// TIA Portal V17 export
// export: Created 2022-07-28T18:02:47.0789834Z, ExportSetting None, DisplayName Totally Integrated Automation Portal, DisplayVersion V17, DisplayName TIA Portal Openness, DisplayVersion V17, DisplayName TIA Portal Teamcenter Gateway, DisplayVersion V17, DisplayName TIA Portal Version Control Interface, DisplayVersion V17, DisplayName TIA Portal Test Suite Advanced, DisplayVersion V17, DisplayName SINAMICS Startdrive Advanced, DisplayVersion V17, DisplayName SINAMICS DCC, DisplayVersion V17, DisplayName SINAMICS Startdrive G130, G150, S120, S150, SINAMICS MV, S210, DisplayVersion V17, DisplayName SINAMICS Startdrive G110M, G120, G120C, G120D, G120P, G115D, DisplayVersion V17, DisplayName STEP 7 Professional, DisplayVersion V17, DisplayName SIMATIC Energy Suite, DisplayVersion V17, DisplayName STEP 7 CFC, DisplayVersion V17, DisplayName STEP 7 Safety, DisplayVersion V17, DisplayName WinCC Advanced / Unified PC, DisplayVersion V17, DisplayName SIMATIC Visualization Architect, DisplayVersion V17
FUNCTION "Outputs_FC" : Void   // FC14, SCL
{ S7_Optimized_Access := 'TRUE' }
// stored: SetENOAutomatically false
BEGIN
   REGION (ID = 1) Витратомір пари на нову рафінацію Steam Flowmeter New
       //Тип елемента: Аналоговий витратомір
       //Параметри давача: Scale=; 4-20mA; Analog = 0 - 27648;
       //Одиниці вимірювання: m3/h
       //Додаткова інформація: SITRANS FX330 / 7ME2610-3LD00-0AA0-Z

   END_REGION

   REGION (ID = 2) Витратомір пари на стару рафінацію Steam Flowmeter Old
       //Тип елемента: Аналоговий витратомір
       //Параметри давача: Scale=; 4-20mA; Analog = 0 - 27648;
       //Одиниці вимірювання: m3/h
       //Додаткова інформація: SITRANS FX330 / 7ME2610-3LD00-0AA0-Z

   END_REGION

   REGION (ID = 3) Перетворювач тиску обор.води PTНГр
       //Тип елемента: Аналоговий сигнал
       //Параметри давача: Scale=0-10bar; 4-20mA; Analog = 0 - 27648;
       //Одиниці вимірювання: bar
       //Додаткова інформація: 

   END_REGION

   REGION (ID = 4) Перетворювач температури вих.води ХМ1 ТТW1011
       //Тип елемента: Аналоговий сигнал
       //Параметри давача: Scale=0-150C; 4-20mA; Analog = 0 - 27648;
       //Одиниці вимірювання: C
       //Додаткова інформація: 

   END_REGION

   REGION (ID = 5) Перетворювач температури вих.води ХМ2 TT811
       //Тип елемента: Аналоговий сигнал
       //Параметри давача: Scale=0-150C; 4-20mA; Analog = 0 - 27648;
       //Одиниці вимірювання: C
       //Додаткова інформація: 

   END_REGION

   REGION (ID = 6) Перетворювач тиску (рівень басейну градирні 1) LTБ1Гр
       //Тип елемента: Аналоговий сигнал
       //Параметри давача: Scale=0-0.25bar; 4-20mA; Analog = 0 - 27648;
       //Одиниці вимірювання: м
       //Додаткова інформація: 

   END_REGION

   REGION (ID = 7) Перетворювач тиску (рівень басейну градирні 2) LTБ2Гр
       //Тип елемента: Аналоговий сигнал
       //Параметри давача: Scale=0-0.25bar; 4-20mA; Analog = 0 - 27648;
       //Одиниці вимірювання: м
       //Додаткова інформація: 

   END_REGION

   REGION (ID = 8) Аналоговий сигнал від AirForce 1 G1
       //Тип елемента: Аналоговий сигнал
       //Параметри давача: Scale= ; 4-20mA; Analog = 0 - 27648;
       //Одиниці вимірювання: 
       //Додаткова інформація: 

   END_REGION

   REGION (ID = 9) Аналоговий сигнал від AirForce 2 G1
       //Тип елемента: Аналоговий сигнал
       //Параметри давача: Scale= ; 4-20mA; Analog = 0 - 27648;
       //Одиниці вимірювання: 
       //Додаткова інформація: 

   END_REGION

   REGION (ID = 10) Аналоговий сигнал від AirForce 3 G1
       //Тип елемента: Аналоговий сигнал
       //Параметри давача: Scale= ; 4-20mA; Analog = 0 - 27648;
       //Одиниці вимірювання: 
       //Додаткова інформація: 

   END_REGION

   REGION (ID = 11) Аналоговий сигнал від AirForce 4 G1
       //Тип елемента: Аналоговий сигнал
       //Параметри давача: Scale= ; 4-20mA; Analog = 0 - 27648;
       //Одиниці вимірювання: 
       //Додаткова інформація: 

   END_REGION

   REGION (ID = 12) Аналоговий сигнал від AirForce 5 G1
       //Тип елемента: Аналоговий сигнал
       //Параметри давача: Scale= ; 4-20mA; Analog = 0 - 27648;
       //Одиниці вимірювання: 
       //Додаткова інформація: 

   END_REGION

   REGION (ID = 13) Аналоговий сигнал від AirForce 6 G1
       //Тип елемента: Аналоговий сигнал
       //Параметри давача: Scale= ; 4-20mA; Analog = 0 - 27648;
       //Одиниці вимірювання: 
       //Додаткова інформація: 

   END_REGION

   REGION (ID = 14) Перетворювач тиску (рівень ємності конденсату) LT R46
       //Тип елемента: Аналоговий сигнал
       //Параметри давача: Scale=0-0.4bar; 4-20mA; Analog = 0 - 27648;
       //Одиниці вимірювання: м
       //Додаткова інформація: 

   END_REGION

   REGION (ID = 15) Температура конденсату TT R46
       //Тип елемента: Аналоговий сигнал
       //Параметри давача: Scale=0-150C; 4-20mA; Analog = 0 - 27648;
       //Одиниці вимірювання: C
       //Додаткова інформація: 

   END_REGION

   REGION (ID = 16) Тиск повітря 1 PT AirLow
       //Тип елемента: Аналоговий сигнал
       //Параметри давача: Scale=0-10bar; 4-20mA; Analog = 0 - 27648;
       //Одиниці вимірювання: bar
       //Додаткова інформація: 

   END_REGION

   REGION (ID = 17) Тиск повітря 2 PT AirHigh
       //Тип елемента: Аналоговий сигнал
       //Параметри давача: Scale=0-10bar; 4-20mA; Analog = 0 - 27648;
       //Одиниці вимірювання: bar
       //Додаткова інформація: 

   END_REGION

   REGION (ID = 18) Тиск газу PT Gas
       //Тип елемента: Аналоговий сигнал
       //Параметри давача: Scale= ;4-20ma; Analog = 0 - 27648;
       //Одиниці вимірювання: 
       //Додаткова інформація: 

   END_REGION

   REGION (ID = 19) Тиск азоту PT Nitrogen
       //Тип елемента: Аналоговий сигнал
       //Параметри давача: Scale= ;4-20ma; Analog = 0 - 27648;
       //Одиниці вимірювання: 
       //Додаткова інформація: 

   END_REGION

   REGION (ID = 20) Тиск води осмотичної PT W10_1
       //Тип елемента: Аналоговий сигнал
       //Параметри давача: Scale=0-6bar; 4-20mA; Analog = 0 - 27648;
       //Одиниці вимірювання: bar
       //Додаткова інформація: 

   END_REGION

   REGION (ID = 21) Тиск води технічної PT water
       //Тип елемента: Аналоговий сигнал
       //Параметри давача: Scale=0-6bar; 4-20mA; Analog = 0 - 27648;
       //Одиниці вимірювання: bar
       //Додаткова інформація: 

   END_REGION

   REGION (ID = 22) Тиск пари 1 PT steam 1
       //Тип елемента: Аналоговий сигнал
       //Параметри давача: Scale= ;4-20ma; Analog = 0 - 27648;
       //Одиниці вимірювання: 
       //Додаткова інформація: 

   END_REGION

   REGION (ID = 23) Тиск пари 2 PT steam 2
       //Тип елемента: Аналоговий сигнал
       //Параметри давача: Scale= ;4-20ma; Analog = 0 - 27648;
       //Одиниці вимірювання: 
       //Додаткова інформація: 

   END_REGION

   REGION (ID = 24) Тиск пари 3 PT steam 3
       //Тип елемента: Аналоговий сигнал
       //Параметри давача: Scale= ;4-20ma; Analog = 0 - 27648;
       //Одиниці вимірювання: 
       //Додаткова інформація: 

   END_REGION

   REGION (ID = 25) Тиск теплоносія 1 PT coolant 1
       //Тип елемента: Аналоговий сигнал
       //Параметри давача: Scale= ;4-20ma; Analog = 0 - 27648;
       //Одиниці вимірювання: 
       //Додаткова інформація: 

   END_REGION

   REGION (ID = 26) Тиск теплоносія 2 PT coolant 2
       //Тип елемента: Аналоговий сигнал
       //Параметри давача: Scale= ;4-20ma; Analog = 0 - 27648;
       //Одиниці вимірювання: 
       //Додаткова інформація: 

   END_REGION

   REGION (ID = 27) Температура теплоносія 1 TT coolant 1
       //Тип елемента: Аналоговий сигнал
       //Параметри давача: Scale=0-150C; 4-20mA; Analog = 0 - 27648;
       //Одиниці вимірювання: C
       //Додаткова інформація: 

   END_REGION

   REGION (ID = 28) Температура теплоносія 2 TT coolant 2
       //Тип елемента: Аналоговий сигнал
       //Параметри давача: Scale=0-150C; 4-20mA; Analog = 0 - 27648;
       //Одиниці вимірювання: C
       //Додаткова інформація: 

   END_REGION

   REGION (ID = 29) Перетворювач тиску подачі  кислоти PT PW579CA
       //Тип елемента: Аналоговий сигнал
       //Параметри давача: Scale=0-6bar; 4-20mA; Analog = 0 - 27648;
       //Одиниці вимірювання: bar
       //Додаткова інформація: 

   END_REGION

   REGION (ID = 30) Рівень в ємності лимонної кислоти LT PW579CA
       //Тип елемента: Аналоговий сигнал
       //Параметри давача: Scale=0-0.1bar; 4-20mA; Analog = 0 - 27648;
       //Одиниці вимірювання: м
       //Додаткова інформація: 

   END_REGION

   REGION (ID = 31) Перетворювач тиску подачі  лугу PT PW579NA
       //Тип елемента: Аналоговий сигнал
       //Параметри давача: Scale=0-6bar; 4-20mA; Analog = 0 - 27648;
       //Одиниці вимірювання: bar
       //Додаткова інформація: 

   END_REGION

   REGION (ID = 32) Перетворювач тиску (рівень води в ємності) LT W10 OW
       //Тип елемента: Аналоговий сигнал
       //Параметри давача: Scale=0-0.25bar; 4-20mA; Analog = 0 - 27648;
       //Одиниці вимірювання: м
       //Додаткова інформація: 

   END_REGION

   REGION (ID = 33) Температура води охолодження дублюючого насоса TT P822 2
       //Тип елемента: Аналоговий сигнал
       //Параметри давача: Scale= ; 4-20mA; Analog = 0 - 27648;
       //Одиниці вимірювання: C
       //Додаткова інформація: 

   END_REGION

   REGION (ID = 34) Рівень води в ємності LT W0 W
       //Тип елемента: Аналоговий сигнал
       //Параметри давача: Scale=0-0.25bar; 4-20mA; Analog = 0 - 27648;
       //Одиниці вимірювання: м
       //Додаткова інформація: 

   END_REGION

   REGION (ID = 35) Перетворювач тиску технологічної води PT PW0 W
       //Тип елемента: Аналоговий сигнал
       //Параметри давача: Scale=0-10bar; 4-20mA; Analog = 0 - 27648;
       //Одиниці вимірювання: bar
       //Додаткова інформація: 

   END_REGION

   REGION (ID = 36) Дискретний сигнал від AirForce 1 G1
       //Тип елемента: Дискретний сигнал
       //Параметри давача: Info;NO;
       //Додаткова інформація: 

   END_REGION

   REGION (ID = 37) Дискретний сигнал від AirForce 2 G1
       //Тип елемента: Дискретний сигнал
       //Параметри давача: Info;NO;
       //Додаткова інформація: 

   END_REGION

   REGION (ID = 38) Дискретний сигнал від AirForce 3 G1
       //Тип елемента: Дискретний сигнал
       //Параметри давача: Info;NO;
       //Додаткова інформація: 

   END_REGION

   REGION (ID = 39) Дискретний сигнал від AirForce 4 G1
       //Тип елемента: Дискретний сигнал
       //Параметри давача: Info;NO;
       //Додаткова інформація: 

   END_REGION

   REGION (ID = 40) Дискретний сигнал від AirForce 5 G1
       //Тип елемента: Дискретний сигнал
       //Параметри давача: Info;NO;
       //Додаткова інформація: 

   END_REGION

   REGION (ID = 41) Контроль роботи холодильної машини 1 - робота W1011
       //Тип елемента: Дискретний сигнал
       //Параметри давача: Info;NO;
       //Додаткова інформація: 

   END_REGION

   REGION (ID = 42) Контроль роботи холодильної машини 1 - аварія W1011
       //Тип елемента: Дискретний сигнал
       //Параметри давача: Err;NO;
       //Додаткова інформація: 

   END_REGION

   REGION (ID = 43) Контроль роботи холодильної машини 2 - робота 811
       //Тип елемента: Дискретний сигнал
       //Параметри давача: Info;NO;
       //Додаткова інформація: 

   END_REGION

   REGION (ID = 44) Контроль роботи холодильної машини 2 - аварія 811
       //Тип елемента: Дискретний сигнал
       //Параметри давача: Err;NO;
       //Додаткова інформація: 

   END_REGION

   REGION (ID = 45) Парогенератор і бойлерна - робота DI7
       //Тип елемента: Дискретний сигнал
       //Параметри давача: Info;NO;
       //Додаткова інформація: 

   END_REGION

   REGION (ID = 46) Парогенератор і бойлерна - аварія DI7
       //Тип елемента: Дискретний сигнал
       //Параметри давача: Err;NC;
       //Додаткова інформація: 

   END_REGION

   REGION (ID = 47) Парогенератор і бойлерна - загазованість DI7
       //Тип елемента: Дискретний сигнал
       //Параметри давача: Err;NC;
       //Додаткова інформація: 

   END_REGION

   REGION (ID = 48) Протік  води охолодження дублюючого насоса FT P822 2
       //Тип елемента: Дискретний сигнал
       //Параметри давача: Info;NC;
       //Додаткова інформація: 

   END_REGION

   REGION (ID = 10) Насос відкачки конденсату 1 PR46 1
       //Тип елемента: Насос без ПЧ
       //Параметри двигуна: P=4.6kW;V=400V;I=8.2A;v=2950rpm;

       "Q_PR46_1_KM" := "D_InOut"."PR46_1".Q_KM_Cmd;
   END_REGION

   REGION (ID = 11) Насос відкачки конденсату 2 PR46 2
       //Тип елемента: Насос без ПЧ
       //Параметри двигуна: P=4.6kW;V=400V;I=8.2A;v=2950rpm;

       "Q_PR46_2_KM" := "D_InOut"."PR46_2".Q_KM_Cmd;
   END_REGION

   REGION (ID = 12) Насос подачі кислоти PW579CA
       //Тип елемента: Насос без ПЧ
       //Параметри двигуна: P=3kW;V=400V;I=6.33A;f=0.79;v=2880rpm;

       "Q_PW579CA_KM" := "D_InOut"."PW579CA".Q_KM_Cmd;
   END_REGION

   REGION (ID = 13) Насос подачі лугу PW579NA
       //Тип елемента: Насос без ПЧ
       //Параметри двигуна: P=3kW;V=400V;I=6.33A;f=0.79;v=2880rpm;

       "Q_PW579NA_KM" := "D_InOut"."PW579NA".Q_KM_Cmd;
   END_REGION

   REGION (ID = 14) Насос оборотної води 1 Н1Гр
       //Тип елемента: Насос з ПЧ
       //Параметри двигуна: P=75kW;V=400V;I=133A;f=0.86;v=2979rpm;
       //Параметри ПЧ: G120C; Profinet = 8 Words;

   END_REGION

   REGION (ID = 15) Насос оборотної води 2 Н2Гр
       //Тип елемента: Насос з ПЧ
       //Параметри двигуна: P=75kW;V=400V;I=133A;f=0.86;v=2979rpm;
       //Параметри ПЧ: G120C; Profinet = 8 Words;

   END_REGION

   REGION (ID = 16) Насос оборотної води 3 Н3Гр
       //Тип елемента: Насос з ПЧ
       //Параметри двигуна: P=75kW;V=400V;I=133A;f=0.86;v=2979rpm;
       //Параметри ПЧ: G120C; Profinet = 8 Words;

   END_REGION

   REGION (ID = 17) Насос подачі технологічної води PW0 W
       //Тип елемента: Насос з ПЧ
       //Параметри двигуна: P=15kW;V=400V;I=A;f=;v=rpm;
       //Параметри ПЧ: G120C; Profinet = 8 Words;

   END_REGION

   REGION (ID = 18) Регулятор температути вихідної води 1 TIC_W1011
       //Тип елемента: ПІД

       "QI_FYW1011_VlvSP" := "D_InOut"."TIC_W1011".QI_AnalogValue;
   END_REGION

   REGION (ID = 19) Регулятор температути вихідної води 2 TIC_811
       //Тип елемента: ПІД

       "QI_FY811_VlvSP" := "D_InOut"."TIC_811".QI_AnalogValue;
   END_REGION

   REGION (ID = 20) Регулятор тиску кислоти LIC_PW579CA
       //Тип елемента: ПІД

       "QI_FY_PW579CA_VlvSP" := "D_InOut"."LIC_PW579CA".QI_AnalogValue;
   END_REGION

   REGION (ID = 21) Регулятор тиску лугу LIC_PW579NA
       //Тип елемента: ПІД

       "QI_FY_PW579NA_VlvSP" :="D_InOut"."LIC_PW579NA".QI_AnalogValue;
   END_REGION

   REGION (ID = 22) Регулятор тиску технологічної води PIC_PW0_W
       //Тип елемента: ПІД

       //"Q_PIC_PW0_W" := "D_InOut"."PIC_PW0_W".QI_AnalogValue;
   END_REGION

   REGION (ID = 23) Регулятор тиску оборотної води PIC_N_Gr
       //Тип елемента: ПІД каскадний

   END_REGION

   REGION (ID = 1) Клапан продувки басейну градирні 1 XVБ1Гр
       //Тип елемента: Клапан продувки

       "Q_XVB1Gr_VlvCmd" := "D_InOut"."XVB1Gr".Cmd_Open;
   END_REGION

   REGION (ID = 2) Клапан підживлення градирні 1 XV1Гр
       //Тип елемента: Клапан двоходовий (Дискретний)

       "Q_XV1Gr_VlvCmd" := "D_InOut"."XV1Gr".Cmd_Open;
   END_REGION

   REGION (ID = 3) Клапан продувки басейну градирні 2 XVБ2Гр
       //Тип елемента: Клапан продувки

       "Q_XVB2Gr_VlvCmd" := "D_InOut"."XVB2Gr".Cmd_Open;
   END_REGION

   REGION (ID = 4) Клапан підживлення градирні 2 XV2Гр
       //Тип елемента: Клапан двоходовий (Дискретний)

       "Q_XV2Gr_VlvCmd" := "D_InOut"."XV2Gr".Cmd_Open;
   END_REGION

   REGION (ID = 5) Клапан подачі конденсату до W578HW1 XV W578HW1/R46
       //Тип елемента: Клапан конденсату

       "Q_XV_W578HW1_R46_VlvCmd" := "D_InOut"."XV_W578HW1_R46".Cmd_Open;
   END_REGION

   REGION (ID = 6) Клапан подачі конденсату до градирні XV Бгр/R46
       //Тип елемента: Клапан конденсату

       "Q_XV_BGr_R46_VlvCmd" := "D_InOut"."XV_BGr_R46".Cmd_Open;
   END_REGION

   REGION (ID = 7) Клапан подачі конденсату до котельні ОЕЗ XV Storage/R46
       //Тип елемента: Клапан конденсату

       "Q_XV_Storage_R46_VlvCmd" := "D_InOut"."XV_Storage_R46".Cmd_Open;
   END_REGION

   REGION (ID = 8) Відсічний клапан XV6
       //Тип елемента: Клапан двоходовий (Дискретний)

       "Q_XV6_Safe_VlvCmd" := "D_InOut"."XV6_Safe".Cmd_Open;
   END_REGION

   REGION (ID = 9) Клапан подачі води в ємність запасу осмотичної води XV W10 OW
       //Тип елемента: Клапан двоходовий (Дискретний)

       "Q_XV_W10_OW_VlvCmd" := "D_InOut"."XV_W10_OW".Cmd_Open;
   END_REGION
END_FUNCTION
